PROGRAM PRG_1_PlcTask
VAR
    fbLogHandler: FB_LogHandler;

 

END_VAR

fbLogHandler();


PRG_2_AT1K4();

END_PROGRAM

(* stored: Version 1.1.0.1, ProductVersion 3.1.4024.3
   POU PRG_1_PlcTask: Id {e5334f36-3c5f-4553-b6cf-4e9240a43836}, SpecialFunc None *)
